TYPE ST_Crop :
STRUCT
	crop_id : INT;
	crop_status : INT;
	level : INT;
	plant_id : INT;
	stack : INT;
	stage : INT;
	plant : ST_PlantConfig;
END_STRUCT
END_TYPE

(* stored: Version 1.1.0.1, ProductVersion 3.1.4024.12
   DUT ST_Crop: Id {e06d4db4-e791-4d31-8613-53ad6e6118b0} *)
